// TIA Portal V20 export
TYPE "typeFDoorSwitchStatus"
// stored: Access Published, IsFailsafeCompliant true, Namespace Safety
   STRUCT
      UnwinderTopDoorOpen : Bool;   // Zone 1 -MAIN (EC Top) gate is opened
      UnwinderLeftDoorOpen : Bool;   // Zone 2 -EC LH roll change gate is opened
      UnwinderRightDoorOpen : Bool;   // Zone 3 -EC RH roll change gate is opened
      CutterDoorOpen : Bool;   // Zone 1 - Cutter gate is opened
      MagazineDoorOpen : Bool;   // Zone 1 - Magazine System gate is opened
      ConveyorDoorOpen : Bool;   // Zone 1 - Conveyror area gate is opened
      ScrapBoxDoorOpen : Bool;   // Zone 1 - Cutter gate is opened
      ScrapBoxDoorClose : Bool;   // Zone 1 - ScrapBox gate is closed
      CentralAisleDoorOpen : Bool;   // Zone 1 - Central Aisle gate is opened
      TotalOneDoorOpen : Bool;   // F Door Open Status
   END_STRUCT;
END_TYPE
